{attribute 'GeneratedUsingTerminal: EL2521-0124-0018'}
{attribute addProperty BoxType "EL2521-0124-0018"}
{attribute addProperty Id "StatusAT %I*Status_B83811715"}
{attribute addProperty CRC "3773501672"}
{attribute addProperty Size "5"}
TYPE PTO_Status_E0EB10E8 :
STRUCT
	{attribute addProperty Name "Status"}
	Status AT %I* : Status_B8381171;
END_STRUCT
END_TYPE

(* stored: Version 1.2.0.0, ProductVersion 3.1.4024.9
   DUT PTO_Status_E0EB10E8: Id {716fa9db-e008-4e07-9081-c8e40a8dc3d5} *)
